# EPICS autosave request: apps/prologixApp/Db/prologix_settings.req
#
# Prologix GPIB-ETHERNET Controller
#
# Author: Wesley Moore
# Date:   July 2015
#

$(P)$(R)ADDR:SET
$(P)$(R)AUTO:SET
$(P)$(R)EOS:SET
$(P)$(R)MODE:SET
$(P)$(R)SAVECFG:SET
